FUNCTION_BLOCK DINT_Param
VAR_INPUT PERSISTENT
	val			: DINT;
END_VAR

END_FUNCTION_BLOCK

(* stored: Version 1.1.0.1
   POU DINT_Param: Id {1a45a280-63f7-4da9-b52a-2940f5b9a706}, SpecialFunc None *)
